FUNCTION F_GetDefaultWoodPanel : ST_WoodPanelData
VAR_INPUT
END_VAR
VAR
END_VAR

F_GetDefaultWoodPanel.rPanelWidth := 100.0; // Default width: 100mm
F_GetDefaultWoodPanel.rPanelLength := 500.0; // Default length: 500mm
F_GetDefaultWoodPanel.rPanelThickness := 5.0; // Default thickness: 5mm

END_FUNCTION

(* stored: Version 1.1.0.1
   POU F_GetDefaultWoodPanel: Id {ec0410ba-a39e-467c-8bf4-d774a2f79cd1}, SpecialFunc None *)
